Omron CX-Programmer project NewProject (CX-Programmer 9.75)

# PLC NewPLC1: CP1E E20

## Program NewProgram1 (cyclic task 0)
Local symbols
GREEN 100.00 BOOL
GREEN_B 100.03 BOOL
GREEN_C 100.06 BOOL
GREEN_D 101.01 BOOL
MAIN 10.00 BOOL
MEM1 10.00 BOOL
MEM2 10.01 BOOL
MEM3 10.02 BOOL
MEM4 10.05 BOOL
RED 100.02 BOOL
RED_B 100.05 BOOL
RED_C 101.00 BOOL
RED_D 101.03 BOOL
START 0.00 BOOL
STOP 0.01 BOOL
YELLOW 100.01 BOOL
YELLOW_B 100.04 BOOL
YELLOW_C 100.07 BOOL
YELLOW_D 101.02 BOOL

### Section Section1

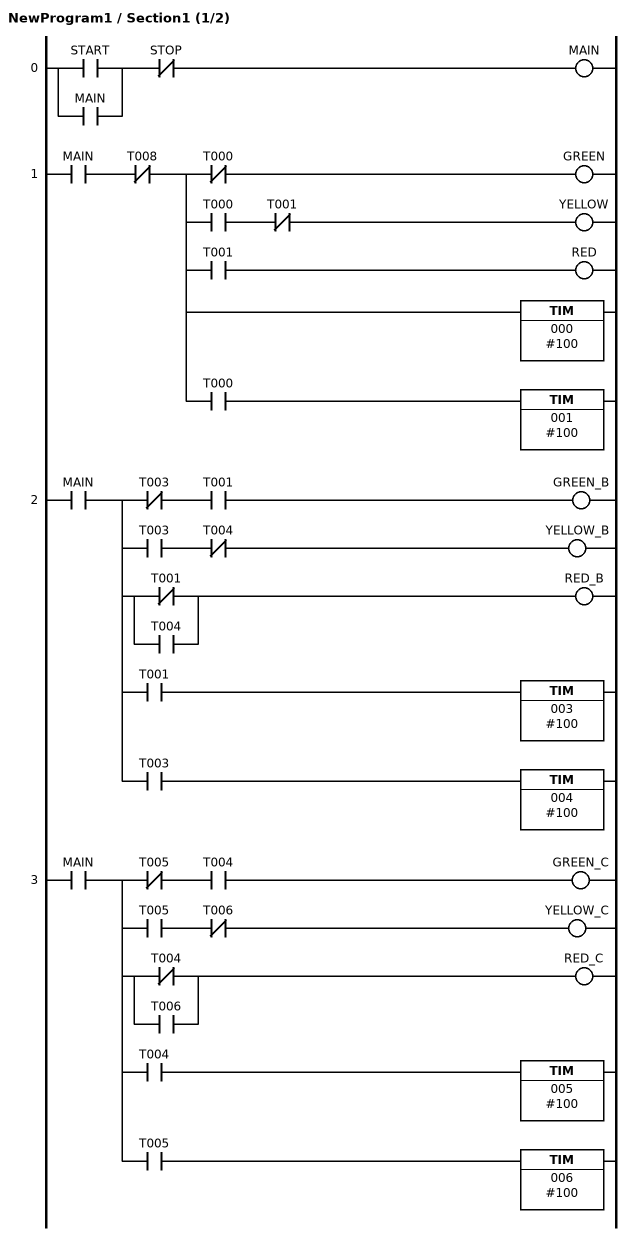
; rung 0
LD START
OR MAIN
ANDNOT STOP
OUT MAIN
; rung 1
LD MAIN
ANDNOT T008
OUT TR0
ANDNOT T000
OUT GREEN
LD TR0
AND T000
ANDNOT T001
OUT YELLOW
LD TR0
AND T001
OUT RED
LD TR0
TIM 000 #100
AND T000
TIM 001 #100
; rung 2
LD MAIN
OUT TR0
ANDNOT T003
AND T001
OUT GREEN_B
LD TR0
AND T003
ANDNOT T004
OUT YELLOW_B
LD TR0
LDNOT T001
OR T004
ANDLD
OUT RED_B
LD TR0
AND T001
TIM 003 #100
LD TR0
AND T003
TIM 004 #100
; rung 3
LD MAIN
OUT TR0
ANDNOT T005
AND T004
OUT GREEN_C
LD TR0
AND T005
ANDNOT T006
OUT YELLOW_C
LD TR0
LDNOT T004
OR T006
ANDLD
OUT RED_C
LD TR0
AND T004
TIM 005 #100
LD TR0
AND T005
TIM 006 #100

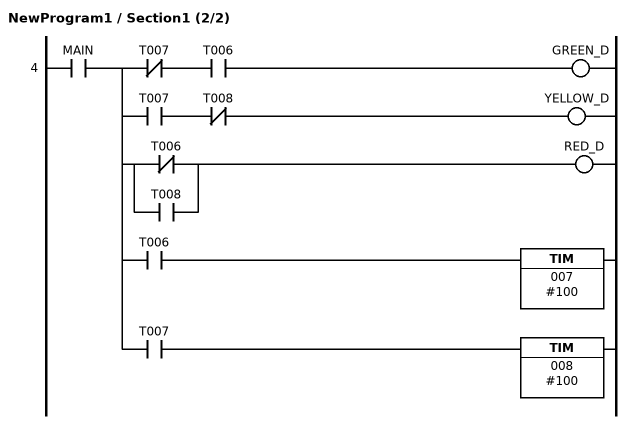
; rung 4
LD MAIN
OUT TR0
ANDNOT T007
AND T006
OUT GREEN_D
LD TR0
AND T007
ANDNOT T008
OUT YELLOW_D
LD TR0
LDNOT T006
OR T008
ANDLD
OUT RED_D
LD TR0
AND T006
TIM 007 #100
LD TR0
AND T007
TIM 008 #100

### Section END
; rung 0
END(001)